// TIA Portal V20 export
DATA_BLOCK "HmiInterface"   // DB95
{ DB_Accessible_From_OPC_UA := 'FALSE' }
AUTHOR : ERsystem_FA2_DH. Kim
// stored: Access Published, DBAccessibleFromOPCUA false, DBAccessibleFromWebserver false, MemoryReserve 100, Namespace Unit1.Em3
   VAR
      em : "LAF_typeEmInterface";
      cm : Struct
         softCam : "Unit1.type_emRelations_em3_SoftCam";
      END_STRUCT;
      webGuide : Struct
         jobs { S7_SetPoint := 'True'} : "LAF_typeJobsInterface";
         sequence { S7_SetPoint := 'True'} : "LAF_typeSequenceInterface";
      END_STRUCT;
      auxiliary : Struct
         cmEpc_UnUse : Bool;
         dancerRegulator : LReal;
      END_STRUCT;
      cmSafetyPinIdlePositionSensor { S7_SetPoint := 'True'} : "LBC_typeDigitalSignalInterface";
      cmRotationSafetyPinPositionSensor { S7_SetPoint := 'True'} : "LBC_typeDigitalSignalInterface";
      cmIonizerTopMaintDetection { S7_SetPoint := 'True'} : "LBC_typeDigitalSignalInterface";
      cmIonizerTopErrorDetection { S7_SetPoint := 'True'} : "LBC_typeDigitalSignalInterface";
      cmIonizerBtmMaintDetection { S7_SetPoint := 'True'} : "LBC_typeDigitalSignalInterface";
      cmIonizerBtmErrorDetection { S7_SetPoint := 'True'} : "LBC_typeDigitalSignalInterface";
      cmDancerEncoder : "LBC_typeAnalogInputInterface";
      cmLoadCellControllerInterface : "LBC_typeAnalogInputInterface";
      cmDancerElectroPneumaticRegulator : "LBC_typeAnalogOutputInterface";
      cmCompensatorAxisX : "LBC_typeAxis64PosInterface";
      cmMasterVirtualAxis { S7_SetPoint := 'True'} : "LBC_typeAxis64PosInterface";
      cmUnwinderVirtualAxis : "LBC_typeAxis64PosInterface";
      cmDancerFwdBwd : "LBC_typeTwoWayActuatorInterface";
      cmSepaUnwinderIonizerTop { S7_SetPoint := 'True'} : "LBC_typeTwoWayActuatorInterface";
      cmSepaUnwinderIonizerBottom { S7_SetPoint := 'True'} : "LBC_typeTwoWayActuatorInterface";
      cmEpcPivot : "LER_typeCON600Interface";
      motion : Struct
         jobs { S7_SetPoint := 'True'} : "LAF_typeJobsInterface";
         sequence { S7_SetPoint := 'True'} : "LAF_typeSequenceInterface";
      END_STRUCT;
      "step" : Struct
         jobs { S7_SetPoint := 'True'} : "LAF_typeJobsInterface";
         sequence { S7_SetPoint := 'True'} : "LAF_typeSequenceInterface";
      END_STRUCT;
      intCondition : Struct
         Axis_03 { S7_SetPoint := 'True'} : "LER.typeAxisIntlockAll";   // compenastor X
         Actuator_10 { S7_SetPoint := 'True'} : "LER.typeAxisActuatorCondition";   // DancerFwdBwd
         Actuator_11 { S7_SetPoint := 'True'} : "LER.typeAxisActuatorCondition";   // SepaUnwinderIonizer
         Actuator_12 { S7_SetPoint := 'True'} : "LER.typeAxisActuatorCondition";   // SepaUnwinderIonizerBottom
      END_STRUCT;
   END_VAR
BEGIN
   em.interlinkMode.link := FALSE;
   em.interlinkMode.unlink := FALSE;
   em.interlinkMode.isLinked := TRUE;
   em.commands.enable := FALSE;
   em.commands.acknowledge := FALSE;
   em.commands.disableAlarms := FALSE;
   em.commands.activateSimulation := FALSE;
   em.commands.home := FALSE;
   em.commands.moveToInitialPosition := FALSE;
   em.commands.directModeControl := 16#0000_0002;
   em.commands.directStateControl := 16#0000_0002;
   em.status.enabled := TRUE;
   em.status.acknowledgeActive := FALSE;
   em.status.alarmsDisabled := FALSE;
   em.status.simulationActive := FALSE;
   em.status.safetyReleased := TRUE;
   em.status.initialized := FALSE;
   em.status.homed := TRUE;
   em.status.safeState := FALSE;
   em.status.stateComplete := TRUE;
   cmSafetyPinIdlePositionSensor.commands.refreshConfiguration := FALSE;
   cmSafetyPinIdlePositionSensor.commands.editConfiguration := FALSE;
   cmSafetyPinIdlePositionSensor.commands.saveConfiguration := FALSE;
   cmSafetyPinIdlePositionSensor.commands.reset := FALSE;
   cmSafetyPinIdlePositionSensor.monitoring.enable := TRUE;
   cmSafetyPinIdlePositionSensor.monitoring.referenceDesignator := WSTRING#'U1.EM3 WebGuide.DigitalSignal';
   cmSafetyPinIdlePositionSensor.monitoring.simulation := FALSE;
   cmSafetyPinIdlePositionSensor.monitoring.processValue := TRUE;
   cmSafetyPinIdlePositionSensor.monitoring.error := FALSE;
   cmSafetyPinIdlePositionSensor.monitoring.status := 16#0000;
   cmSafetyPinIdlePositionSensor.configuration.referenceDesignator := WSTRING#'DigitalSignal';
   cmSafetyPinIdlePositionSensor.configuration.onDelay := T#0MS;
   cmSafetyPinIdlePositionSensor.configuration.offDelay := T#0MS;
   cmSafetyPinIdlePositionSensor.configuration.default := FALSE;
   cmSafetyPinIdlePositionSensor.configuration.invertProcessValue := FALSE;
   cmSafetyPinIdlePositionSensor.configuration.disableAlarms := FALSE;
   cmRotationSafetyPinPositionSensor.commands.refreshConfiguration := FALSE;
   cmRotationSafetyPinPositionSensor.commands.editConfiguration := FALSE;
   cmRotationSafetyPinPositionSensor.commands.saveConfiguration := FALSE;
   cmRotationSafetyPinPositionSensor.commands.reset := FALSE;
   cmRotationSafetyPinPositionSensor.monitoring.enable := TRUE;
   cmRotationSafetyPinPositionSensor.monitoring.referenceDesignator := WSTRING#'U1.EM3 WebGuide.DigitalSignal';
   cmRotationSafetyPinPositionSensor.monitoring.simulation := FALSE;
   cmRotationSafetyPinPositionSensor.monitoring.processValue := TRUE;
   cmRotationSafetyPinPositionSensor.monitoring.error := FALSE;
   cmRotationSafetyPinPositionSensor.monitoring.status := 16#0000;
   cmRotationSafetyPinPositionSensor.configuration.referenceDesignator := WSTRING#'DigitalSignal';
   cmRotationSafetyPinPositionSensor.configuration.onDelay := T#0MS;
   cmRotationSafetyPinPositionSensor.configuration.offDelay := T#0MS;
   cmRotationSafetyPinPositionSensor.configuration.default := FALSE;
   cmRotationSafetyPinPositionSensor.configuration.invertProcessValue := FALSE;
   cmRotationSafetyPinPositionSensor.configuration.disableAlarms := FALSE;
   cmIonizerTopMaintDetection.commands.refreshConfiguration := FALSE;
   cmIonizerTopMaintDetection.commands.editConfiguration := FALSE;
   cmIonizerTopMaintDetection.commands.saveConfiguration := FALSE;
   cmIonizerTopMaintDetection.commands.reset := FALSE;
   cmIonizerTopMaintDetection.monitoring.enable := TRUE;
   cmIonizerTopMaintDetection.monitoring.referenceDesignator := WSTRING#'U1.EM3 WebGuide.DigitalSignal';
   cmIonizerTopMaintDetection.monitoring.simulation := FALSE;
   cmIonizerTopMaintDetection.monitoring.processValue := FALSE;
   cmIonizerTopMaintDetection.monitoring.error := FALSE;
   cmIonizerTopMaintDetection.monitoring.status := 16#0000;
   cmIonizerTopMaintDetection.configuration.referenceDesignator := WSTRING#'DigitalSignal';
   cmIonizerTopMaintDetection.configuration.onDelay := T#0MS;
   cmIonizerTopMaintDetection.configuration.offDelay := T#0MS;
   cmIonizerTopMaintDetection.configuration.default := FALSE;
   cmIonizerTopMaintDetection.configuration.invertProcessValue := FALSE;
   cmIonizerTopMaintDetection.configuration.disableAlarms := FALSE;
   cmIonizerTopErrorDetection.commands.refreshConfiguration := FALSE;
   cmIonizerTopErrorDetection.commands.editConfiguration := FALSE;
   cmIonizerTopErrorDetection.commands.saveConfiguration := FALSE;
   cmIonizerTopErrorDetection.commands.reset := FALSE;
   cmIonizerTopErrorDetection.monitoring.enable := TRUE;
   cmIonizerTopErrorDetection.monitoring.referenceDesignator := WSTRING#'U1.EM3 WebGuide.DigitalSignal';
   cmIonizerTopErrorDetection.monitoring.simulation := FALSE;
   cmIonizerTopErrorDetection.monitoring.processValue := TRUE;
   cmIonizerTopErrorDetection.monitoring.error := FALSE;
   cmIonizerTopErrorDetection.monitoring.status := 16#0000;
   cmIonizerTopErrorDetection.configuration.referenceDesignator := WSTRING#'DigitalSignal';
   cmIonizerTopErrorDetection.configuration.onDelay := T#0MS;
   cmIonizerTopErrorDetection.configuration.offDelay := T#0MS;
   cmIonizerTopErrorDetection.configuration.default := FALSE;
   cmIonizerTopErrorDetection.configuration.invertProcessValue := FALSE;
   cmIonizerTopErrorDetection.configuration.disableAlarms := FALSE;
   cmIonizerBtmMaintDetection.commands.refreshConfiguration := FALSE;
   cmIonizerBtmMaintDetection.commands.editConfiguration := FALSE;
   cmIonizerBtmMaintDetection.commands.saveConfiguration := FALSE;
   cmIonizerBtmMaintDetection.commands.reset := FALSE;
   cmIonizerBtmMaintDetection.monitoring.enable := TRUE;
   cmIonizerBtmMaintDetection.monitoring.referenceDesignator := WSTRING#'U1.EM3 WebGuide.DigitalSignal';
   cmIonizerBtmMaintDetection.monitoring.simulation := FALSE;
   cmIonizerBtmMaintDetection.monitoring.processValue := FALSE;
   cmIonizerBtmMaintDetection.monitoring.error := FALSE;
   cmIonizerBtmMaintDetection.monitoring.status := 16#0000;
   cmIonizerBtmMaintDetection.configuration.referenceDesignator := WSTRING#'DigitalSignal';
   cmIonizerBtmMaintDetection.configuration.onDelay := T#0MS;
   cmIonizerBtmMaintDetection.configuration.offDelay := T#0MS;
   cmIonizerBtmMaintDetection.configuration.default := FALSE;
   cmIonizerBtmMaintDetection.configuration.invertProcessValue := FALSE;
   cmIonizerBtmMaintDetection.configuration.disableAlarms := FALSE;
   cmIonizerBtmErrorDetection.commands.refreshConfiguration := FALSE;
   cmIonizerBtmErrorDetection.commands.editConfiguration := FALSE;
   cmIonizerBtmErrorDetection.commands.saveConfiguration := FALSE;
   cmIonizerBtmErrorDetection.commands.reset := FALSE;
   cmIonizerBtmErrorDetection.monitoring.enable := TRUE;
   cmIonizerBtmErrorDetection.monitoring.referenceDesignator := WSTRING#'U1.EM3 WebGuide.DigitalSignal';
   cmIonizerBtmErrorDetection.monitoring.simulation := FALSE;
   cmIonizerBtmErrorDetection.monitoring.processValue := TRUE;
   cmIonizerBtmErrorDetection.monitoring.error := FALSE;
   cmIonizerBtmErrorDetection.monitoring.status := 16#0000;
   cmIonizerBtmErrorDetection.configuration.referenceDesignator := WSTRING#'DigitalSignal';
   cmIonizerBtmErrorDetection.configuration.onDelay := T#0MS;
   cmIonizerBtmErrorDetection.configuration.offDelay := T#0MS;
   cmIonizerBtmErrorDetection.configuration.default := FALSE;
   cmIonizerBtmErrorDetection.configuration.invertProcessValue := FALSE;
   cmIonizerBtmErrorDetection.configuration.disableAlarms := FALSE;
   cmDancerEncoder.commands.refreshConfiguration := FALSE;
   cmDancerEncoder.commands.editConfiguration := FALSE;
   cmDancerEncoder.commands.saveConfiguration := FALSE;
   cmDancerEncoder.commands.reset := FALSE;
   cmDancerEncoder.monitoring.enable := TRUE;
   cmDancerEncoder.monitoring.referenceDesignator := WSTRING#'U1.EM3 WebGuide.cmDancerEncoder';
   cmDancerEncoder.monitoring.simulation := FALSE;
   cmDancerEncoder.monitoring.processValue := 0.034215856481481;
   cmDancerEncoder.monitoring.analogValue := 13835;
   cmDancerEncoder.monitoring.limitHigh2 := FALSE;
   cmDancerEncoder.monitoring.limitHigh1 := FALSE;
   cmDancerEncoder.monitoring.limitLow1 := FALSE;
   cmDancerEncoder.monitoring.limitLow2 := FALSE;
   cmDancerEncoder.monitoring.maxValueReached := FALSE;
   cmDancerEncoder.monitoring.minValueReached := FALSE;
   cmDancerEncoder.monitoring.error := FALSE;
   cmDancerEncoder.monitoring.status := 16#0000;
   cmDancerEncoder.configuration.referenceDesignator := WSTRING#'cmDancerEncoder';
   cmDancerEncoder.configuration.physicalUnit := 'unit';
   cmDancerEncoder.configuration.isUnipolarSignal := TRUE;
   cmDancerEncoder.configuration.default := 0.0;
   cmDancerEncoder.configuration.limitHigh2 := 20.0;
   cmDancerEncoder.configuration.limitHigh1 := 15.0;
   cmDancerEncoder.configuration.limitLow1 := -15.0;
   cmDancerEncoder.configuration.limitLow2 := -20.0;
   cmDancerEncoder.configuration.processValueMax := 43.0;
   cmDancerEncoder.configuration.processValueMin := -43.0;
   cmDancerEncoder.configuration.scaleAnalogUppPoint := 27648.0;
   cmDancerEncoder.configuration.scaleAnalogLowPoint := 0.0;
   cmDancerEncoder.configuration.scaleProcessUppPoint := 43.0;
   cmDancerEncoder.configuration.scaleProcessLowPoint := -43.0;
   cmDancerEncoder.configuration.disableAlarms := FALSE;
   cmLoadCellControllerInterface.commands.refreshConfiguration := FALSE;
   cmLoadCellControllerInterface.commands.editConfiguration := FALSE;
   cmLoadCellControllerInterface.commands.saveConfiguration := FALSE;
   cmLoadCellControllerInterface.commands.reset := FALSE;
   cmLoadCellControllerInterface.monitoring.enable := TRUE;
   cmLoadCellControllerInterface.monitoring.referenceDesignator := WSTRING#'U1.EM3 WebGuide.cmLoadCellController';
   cmLoadCellControllerInterface.monitoring.simulation := FALSE;
   cmLoadCellControllerInterface.monitoring.processValue := -99.9638310185185;
   cmLoadCellControllerInterface.monitoring.analogValue := 5;
   cmLoadCellControllerInterface.monitoring.limitHigh2 := FALSE;
   cmLoadCellControllerInterface.monitoring.limitHigh1 := FALSE;
   cmLoadCellControllerInterface.monitoring.limitLow1 := TRUE;
   cmLoadCellControllerInterface.monitoring.limitLow2 := TRUE;
   cmLoadCellControllerInterface.monitoring.maxValueReached := FALSE;
   cmLoadCellControllerInterface.monitoring.minValueReached := FALSE;
   cmLoadCellControllerInterface.monitoring.error := FALSE;
   cmLoadCellControllerInterface.monitoring.status := 16#0000;
   cmLoadCellControllerInterface.configuration.referenceDesignator := WSTRING#'cmLoadCellController';
   cmLoadCellControllerInterface.configuration.physicalUnit := 'unit';
   cmLoadCellControllerInterface.configuration.isUnipolarSignal := TRUE;
   cmLoadCellControllerInterface.configuration.default := 0.0;
   cmLoadCellControllerInterface.configuration.limitHigh2 := 90.0;
   cmLoadCellControllerInterface.configuration.limitHigh1 := 80.0;
   cmLoadCellControllerInterface.configuration.limitLow1 := -80.0;
   cmLoadCellControllerInterface.configuration.limitLow2 := -90.0;
   cmLoadCellControllerInterface.configuration.processValueMax := 100.0;
   cmLoadCellControllerInterface.configuration.processValueMin := -100.0;
   cmLoadCellControllerInterface.configuration.scaleAnalogUppPoint := 27648.0;
   cmLoadCellControllerInterface.configuration.scaleAnalogLowPoint := 0.0;
   cmLoadCellControllerInterface.configuration.scaleProcessUppPoint := 100.0;
   cmLoadCellControllerInterface.configuration.scaleProcessLowPoint := -100.0;
   cmLoadCellControllerInterface.configuration.disableAlarms := TRUE;
   cmDancerElectroPneumaticRegulator.commands.refreshConfiguration := FALSE;
   cmDancerElectroPneumaticRegulator.commands.editConfiguration := FALSE;
   cmDancerElectroPneumaticRegulator.commands.saveConfiguration := FALSE;
   cmDancerElectroPneumaticRegulator.commands.reset := FALSE;
   cmDancerElectroPneumaticRegulator.monitoring.enable := TRUE;
   cmDancerElectroPneumaticRegulator.monitoring.referenceDesignator := WSTRING#'cmDancerRegulator';
   cmDancerElectroPneumaticRegulator.monitoring.simulation := FALSE;
   cmDancerElectroPneumaticRegulator.monitoring.processValue := 0.0;
   cmDancerElectroPneumaticRegulator.monitoring.analogValue := 0;
   cmDancerElectroPneumaticRegulator.monitoring.limitHigh2 := FALSE;
   cmDancerElectroPneumaticRegulator.monitoring.limitHigh1 := FALSE;
   cmDancerElectroPneumaticRegulator.monitoring.limitLow1 := TRUE;
   cmDancerElectroPneumaticRegulator.monitoring.limitLow2 := TRUE;
   cmDancerElectroPneumaticRegulator.monitoring.maxValueReached := FALSE;
   cmDancerElectroPneumaticRegulator.monitoring.minValueReached := FALSE;
   cmDancerElectroPneumaticRegulator.monitoring.error := FALSE;
   cmDancerElectroPneumaticRegulator.monitoring.status := 16#0000;
   cmDancerElectroPneumaticRegulator.configuration.referenceDesignator := WSTRING#'cmDancerRegulator';
   cmDancerElectroPneumaticRegulator.configuration.physicalUnit := 'unit';
   cmDancerElectroPneumaticRegulator.configuration.isUnipolarSignal := TRUE;
   cmDancerElectroPneumaticRegulator.configuration.default := 0;
   cmDancerElectroPneumaticRegulator.configuration.limitHigh2 := 0.5;
   cmDancerElectroPneumaticRegulator.configuration.limitHigh1 := 0.5;
   cmDancerElectroPneumaticRegulator.configuration.limitLow1 := 0.0;
   cmDancerElectroPneumaticRegulator.configuration.limitLow2 := 0.0;
   cmDancerElectroPneumaticRegulator.configuration.processValueMax := 0.5;
   cmDancerElectroPneumaticRegulator.configuration.processValueMin := 0.0;
   cmDancerElectroPneumaticRegulator.configuration.scaleProcessUppPoint := 0.5;
   cmDancerElectroPneumaticRegulator.configuration.scaleProcessLowPoint := 0.0;
   cmDancerElectroPneumaticRegulator.configuration.scaleAnalogUppPoint := 27648.0;
   cmDancerElectroPneumaticRegulator.configuration.scaleAnalogLowPoint := 0.0;
   cmDancerElectroPneumaticRegulator.configuration.disableAlarms := TRUE;
   cmCompensatorAxisX.commandConfiguration.generalSettings.stopOnError := TRUE;
   cmCompensatorAxisX.commandConfiguration.generalSettings.resetWithRestart := FALSE;
   cmCompensatorAxisX.commandConfiguration.generalSettings.abortWaitingSyncCmd := TRUE;
   cmCompensatorAxisX.commandConfiguration.power.startMode := 1;
   cmCompensatorAxisX.commandConfiguration.power.stopMode := 0;
   cmCompensatorAxisX.commandConfiguration.power.syncMotionSimulation := FALSE;
   cmCompensatorAxisX.commandConfiguration.power.syncMotionSimulationExtendedMode := -1;
   cmCompensatorAxisX.commandConfiguration.jog.velocity := 10.0;
   cmCompensatorAxisX.commandConfiguration.jog.acceleration := 100.0;
   cmCompensatorAxisX.commandConfiguration.jog.deceleration := 100.0;
   cmCompensatorAxisX.commandConfiguration.jog.jerk := -1.0;
   cmCompensatorAxisX.commandConfiguration.jog.positionControlled := TRUE;
   cmCompensatorAxisX.commandConfiguration.jog.increment := 0.0;
   cmCompensatorAxisX.commandConfiguration.jog.mode := 0;
   cmCompensatorAxisX.commandConfiguration.moveVelocity.velocity := 10.0;
   cmCompensatorAxisX.commandConfiguration.moveVelocity.acceleration := 100.0;
   cmCompensatorAxisX.commandConfiguration.moveVelocity.deceleration := 100.0;
   cmCompensatorAxisX.commandConfiguration.moveVelocity.jerk := -1.0;
   cmCompensatorAxisX.commandConfiguration.moveVelocity.direction := 0;
   cmCompensatorAxisX.commandConfiguration.moveVelocity.positionControlled := TRUE;
   cmCompensatorAxisX.commandConfiguration.moveVelocity.velocityChangeOnTheFly := FALSE;
   cmCompensatorAxisX.commandConfiguration.stop.deceleration := -1.0;
   cmCompensatorAxisX.commandConfiguration.stop.jerk := -1.0;
   cmCompensatorAxisX.commandConfiguration.stop.abortAcceleration := FALSE;
   cmCompensatorAxisX.commandConfiguration.fastStop.deceleration := -1.0;
   cmCompensatorAxisX.commandConfiguration.fastStop.jerk := -1.0;
   cmCompensatorAxisX.commandConfiguration.fastStop.abortAcceleration := FALSE;
   cmCompensatorAxisX.commandConfiguration.fastStop.replaceStopPossible := FALSE;
   cmCompensatorAxisX.commandConfiguration.torqueLimiting.limit := -1.0;
   cmCompensatorAxisX.commandConfiguration.torqueLimiting.mode := 0;
   cmCompensatorAxisX.commandConfiguration.homing.position := 0.0;
   cmCompensatorAxisX.commandConfiguration.homing.mode := 0;
   cmCompensatorAxisX.commandConfiguration.homing.sensor := 0;
   cmCompensatorAxisX.commandConfiguration.homing.extendedMode := -1;
   cmCompensatorAxisX.commandConfiguration.homing.extendedModeTorqueLimit := 0.0;
   cmCompensatorAxisX.commandConfiguration.homing.extendedModeTargetPosition := 0.0;
   cmCompensatorAxisX.commandConfiguration.posRelative.distance := 0.0;
   cmCompensatorAxisX.commandConfiguration.posRelative.velocity := 10.0;
   cmCompensatorAxisX.commandConfiguration.posRelative.acceleration := 100.0;
   cmCompensatorAxisX.commandConfiguration.posRelative.deceleration := 100.0;
   cmCompensatorAxisX.commandConfiguration.posRelative.jerk := -1.0;
   cmCompensatorAxisX.commandConfiguration.posRelative.direction := 0;
   cmCompensatorAxisX.commandConfiguration.posAbsolute.position := 0.0;
   cmCompensatorAxisX.commandConfiguration.posAbsolute.velocity := 0.0;
   cmCompensatorAxisX.commandConfiguration.posAbsolute.acceleration := -1.0;
   cmCompensatorAxisX.commandConfiguration.posAbsolute.deceleration := -1.0;
   cmCompensatorAxisX.commandConfiguration.posAbsolute.jerk := 57.5863648889861;
   cmCompensatorAxisX.commandConfiguration.posAbsolute.direction := 1;
   cmCompensatorAxisX.commandConfiguration.posAbsolute.positionChangeOnTheFly := FALSE;
   cmCompensatorAxisX.commandConfiguration.posAbsolute.velocityChangeOnTheFly := FALSE;
   cmCompensatorAxisX.commandConfiguration.posSuperimposed.distance := 150.5;
   cmCompensatorAxisX.commandConfiguration.posSuperimposed.velocityDiff := 53.921568627451;
   cmCompensatorAxisX.commandConfiguration.posSuperimposed.acceleration := 31.7185697808535;
   cmCompensatorAxisX.commandConfiguration.posSuperimposed.deceleration := 31.7185697808535;
   cmCompensatorAxisX.commandConfiguration.posSuperimposed.jerk := 18.6579822240315;
   cmCompensatorAxisX.commandConfiguration.posSuperimposed.direction := 0;
   cmCompensatorAxisX.commandConfiguration.haltSuperimposed.deceleration := -1.0;
   cmCompensatorAxisX.commandConfiguration.haltSuperimposed.jerk := -1.0;
   cmCompensatorAxisX.commandConfiguration.haltSuperimposed.abortAcceleration := FALSE;
   cmCompensatorAxisX.commandConfiguration.gearInRelative.ratioNumerator := 10000;
   cmCompensatorAxisX.commandConfiguration.gearInRelative.ratioDenominator := 10000;
   cmCompensatorAxisX.commandConfiguration.gearInRelative.acceleration := -1.0;
   cmCompensatorAxisX.commandConfiguration.gearInRelative.deceleration := -1.0;
   cmCompensatorAxisX.commandConfiguration.gearInRelative.jerk := -1.0;
   cmCompensatorAxisX.commandConfiguration.gearInRelative.ratioChangeOnTheFly := FALSE;
   cmCompensatorAxisX.commandConfiguration.gearInAbsolute.ratioNumerator := 1;
   cmCompensatorAxisX.commandConfiguration.gearInAbsolute.ratioDenominator := 1;
   cmCompensatorAxisX.commandConfiguration.gearInAbsolute.masterSyncPosition := 0.0;
   cmCompensatorAxisX.commandConfiguration.gearInAbsolute.slaveSyncPosition := 0.0;
   cmCompensatorAxisX.commandConfiguration.gearInAbsolute.syncProfileReference := 1;
   cmCompensatorAxisX.commandConfiguration.gearInAbsolute.masterStartDistance := 0.0;
   cmCompensatorAxisX.commandConfiguration.gearInAbsolute.velocity := -1.0;
   cmCompensatorAxisX.commandConfiguration.gearInAbsolute.acceleration := -1.0;
   cmCompensatorAxisX.commandConfiguration.gearInAbsolute.deceleration := -1.0;
   cmCompensatorAxisX.commandConfiguration.gearInAbsolute.jerk := -1.0;
   cmCompensatorAxisX.commandConfiguration.gearInAbsolute.syncDirection := 1;
   cmCompensatorAxisX.commandConfiguration.gearInAbsolute.ratioChangeOnTheFly := FALSE;
   cmCompensatorAxisX.commandConfiguration.gearInVelocity.continuousUpdate := FALSE;
   cmCompensatorAxisX.commandConfiguration.gearInVelocity.ratioNumerator := 1;
   cmCompensatorAxisX.commandConfiguration.gearInVelocity.ratioDenominator := 1;
   cmCompensatorAxisX.commandConfiguration.gearInVelocity.acceleration := -1.0;
   cmCompensatorAxisX.commandConfiguration.gearInVelocity.deceleration := -1.0;
   cmCompensatorAxisX.commandConfiguration.gearInVelocity.jerk := -1.0;
   cmCompensatorAxisX.commandConfiguration.gearInVelocity.positionControlled := FALSE;
   cmCompensatorAxisX.commandConfiguration.camIn.masterOffset := 0.0;
   cmCompensatorAxisX.commandConfiguration.camIn.slaveOffset := 0.0;
   cmCompensatorAxisX.commandConfiguration.camIn.masterScaling := 1.0;
   cmCompensatorAxisX.commandConfiguration.camIn.slaveScaling := 1.0;
   cmCompensatorAxisX.commandConfiguration.camIn.masterSyncPosition := 0.0;
   cmCompensatorAxisX.commandConfiguration.camIn.syncProfileReference := 2;
   cmCompensatorAxisX.commandConfiguration.camIn.masterStartDistance := 0.0;
   cmCompensatorAxisX.commandConfiguration.camIn.velocity := 179.738562091503;
   cmCompensatorAxisX.commandConfiguration.camIn.acceleration := 176.214276560297;
   cmCompensatorAxisX.commandConfiguration.camIn.deceleration := 176.214276560297;
   cmCompensatorAxisX.commandConfiguration.camIn.jerk := 172.759094666958;
   cmCompensatorAxisX.commandConfiguration.camIn.applicationMode := 0;
   cmCompensatorAxisX.commandConfiguration.camIn.syncDirection := 3;
   cmCompensatorAxisX.commandConfiguration.gearOutCamOut.slavePosition := 0.0;
   cmCompensatorAxisX.commandConfiguration.gearOutCamOut.syncProfileReference := 1;
   cmCompensatorAxisX.commandConfiguration.gearOutCamOut.masterStopDistance := 0.0;
   cmCompensatorAxisX.commandConfiguration.gearOutCamOut.deceleration := -1.0;
   cmCompensatorAxisX.commandConfiguration.gearOutCamOut.jerk := -1.0;
   cmCompensatorAxisX.commandConfiguration.gearOutCamOut.syncOutDirection := 3;
   cmCompensatorAxisX.commandConfiguration.gearOutCamOut.gearOutCamOutMode := -1;
   cmCompensatorAxisX.commandConfiguration.phasing.phaseShift := 301.0;
   cmCompensatorAxisX.commandConfiguration.phasing.velocity := 89.8692810457516;
   cmCompensatorAxisX.commandConfiguration.phasing.acceleration := 88.1071382801487;
   cmCompensatorAxisX.commandConfiguration.phasing.deceleration := 88.1071382801487;
   cmCompensatorAxisX.commandConfiguration.phasing.jerk := 0.0;
   cmCompensatorAxisX.commandConfiguration.phasing.profileReference := 0;
   cmCompensatorAxisX.commandConfiguration.phasing.phasingDistance := 0.0;
   cmCompensatorAxisX.commandConfiguration.phasing.startPosition := 45.0;
   cmCompensatorAxisX.commandConfiguration.phasing.direction := 3;
   cmCompensatorAxisX.commandConfiguration.phasing.phaseAbsolute := FALSE;
   cmCompensatorAxisX.commandConfiguration.phasing.phaseShiftChangeOnTheFly := FALSE;
   cmCompensatorAxisX.commandConfiguration.offset.offset := 0.0;
   cmCompensatorAxisX.commandConfiguration.offset.profileReference := 1;
   cmCompensatorAxisX.commandConfiguration.offset.offsetDistance := 0.0;
   cmCompensatorAxisX.commandConfiguration.offset.startPosition := 0.0;
   cmCompensatorAxisX.commandConfiguration.offset.direction := 3;
   cmCompensatorAxisX.commandConfiguration.offset.offsetAbsolute := TRUE;
   cmCompensatorAxisX.commandConfiguration.offset.offsetChangeOnTheFly := FALSE;
   cmCompensatorAxisX.commands.enableMasterControl := FALSE;
   cmCompensatorAxisX.commands.enableAxis := TRUE;
   cmCompensatorAxisX.commands.resetAxis := FALSE;
   cmCompensatorAxisX.commands.openBrake := FALSE;
   cmCompensatorAxisX.commands.jogForward := FALSE;
   cmCompensatorAxisX.commands.jogBackward := FALSE;
   cmCompensatorAxisX.commands.moveVelocity := FALSE;
   cmCompensatorAxisX.commands.stop := FALSE;
   cmCompensatorAxisX.commands.fastStop := FALSE;
   cmCompensatorAxisX.commands.torqueLimiting := FALSE;
   cmCompensatorAxisX.commands.homing := FALSE;
   cmCompensatorAxisX.commands.posRelative := FALSE;
   cmCompensatorAxisX.commands.posAbsolute := FALSE;
   cmCompensatorAxisX.commands.posSuperimposed := FALSE;
   cmCompensatorAxisX.commands.haltSuperimposed := FALSE;
   cmCompensatorAxisX.commands.selectSetPosition := -1;
   cmCompensatorAxisX.commands.uploadParameters := FALSE;
   cmCompensatorAxisX.commands.refreshConfiguration := FALSE;
   cmCompensatorAxisX.commands.editConfiguration := FALSE;
   cmCompensatorAxisX.commands.saveConfiguration := FALSE;
   cmCompensatorAxisX.commands.uploadCurrentTorque := FALSE;
   cmCompensatorAxisX.commands.reset := FALSE;
   cmCompensatorAxisX.monitoring.enable := TRUE;
   cmCompensatorAxisX.monitoring.referenceDesignator := WSTRING#'U1.EM3 WebGuide.cmCompensatorAxisX';
   cmCompensatorAxisX.monitoring.enabled := TRUE;
   cmCompensatorAxisX.monitoring.enableManualCmds := TRUE;
   cmCompensatorAxisX.monitoring.reset := FALSE;
   cmCompensatorAxisX.monitoring.resetAxis := FALSE;
   cmCompensatorAxisX.monitoring.enableAxis := TRUE;
   cmCompensatorAxisX.monitoring.openBrake := FALSE;
   cmCompensatorAxisX.monitoring.jogBackward := FALSE;
   cmCompensatorAxisX.monitoring.jogForward := FALSE;
   cmCompensatorAxisX.monitoring.moveVelocity := FALSE;
   cmCompensatorAxisX.monitoring.stop := FALSE;
   cmCompensatorAxisX.monitoring.fastStop := FALSE;
   cmCompensatorAxisX.monitoring.torqueLimiting := FALSE;
   cmCompensatorAxisX.monitoring.homing := FALSE;
   cmCompensatorAxisX.monitoring.posRelative := FALSE;
   cmCompensatorAxisX.monitoring.posAbsolute := FALSE;
   cmCompensatorAxisX.monitoring.posSuperimposed := FALSE;
   cmCompensatorAxisX.monitoring.haltSuperimposed := FALSE;
   cmCompensatorAxisX.monitoring.brakeOpened := FALSE;
   cmCompensatorAxisX.monitoring.axisEnabled := TRUE;
   cmCompensatorAxisX.monitoring.resetActive := FALSE;
   cmCompensatorAxisX.monitoring.inVelocity := FALSE;
   cmCompensatorAxisX.monitoring.inLimitation := FALSE;
   cmCompensatorAxisX.monitoring.inClamping := FALSE;
   cmCompensatorAxisX.monitoring.startSync := FALSE;
   cmCompensatorAxisX.monitoring.inSync := FALSE;
   cmCompensatorAxisX.monitoring.inSimulation := FALSE;
   cmCompensatorAxisX.monitoring.jogSelected := FALSE;
   cmCompensatorAxisX.monitoring.moveVelocitySelected := FALSE;
   cmCompensatorAxisX.monitoring.stopSelected := FALSE;
   cmCompensatorAxisX.monitoring.fastStopSelected := FALSE;
   cmCompensatorAxisX.monitoring.torqueLimitingSelected := FALSE;
   cmCompensatorAxisX.monitoring.homingSelected := FALSE;
   cmCompensatorAxisX.monitoring.posRelativeSelected := FALSE;
   cmCompensatorAxisX.monitoring.posAbsoluteSelected := FALSE;
   cmCompensatorAxisX.monitoring.posSuperimposedSelected := FALSE;
   cmCompensatorAxisX.monitoring.haltSuperimposedSelected := FALSE;
   cmCompensatorAxisX.monitoring.commandBusy := FALSE;
   cmCompensatorAxisX.monitoring.commandDone := FALSE;
   cmCompensatorAxisX.monitoring.commandAborted := FALSE;
   cmCompensatorAxisX.monitoring.homingCommandBusy := FALSE;
   cmCompensatorAxisX.monitoring.homingCommandDone := FALSE;
   cmCompensatorAxisX.monitoring.homingCommandAborted := FALSE;
   cmCompensatorAxisX.monitoring.superimposedBusy := FALSE;
   cmCompensatorAxisX.monitoring.superimposedDone := FALSE;
   cmCompensatorAxisX.monitoring.superimposedAborted := FALSE;
   cmCompensatorAxisX.monitoring.selectSetPosition := -1;
   cmCompensatorAxisX.monitoring.selectionController := FALSE;
   cmCompensatorAxisX.monitoring.interlockGeneral := TRUE;
   cmCompensatorAxisX.monitoring.interlockJogForward := TRUE;
   cmCompensatorAxisX.monitoring.interlockJogBackward := TRUE;
   cmCompensatorAxisX.monitoring.interlockWarningGeneral := FALSE;
   cmCompensatorAxisX.monitoring.interlockWarningJogForward := FALSE;
   cmCompensatorAxisX.monitoring.interlockWarningJogBackward := FALSE;
   cmCompensatorAxisX.monitoring.valid := TRUE;
   cmCompensatorAxisX.monitoring.busy := TRUE;
   cmCompensatorAxisX.monitoring.error := FALSE;
   cmCompensatorAxisX.monitoring.status := 16#7002;
   cmCompensatorAxisX.monitoring.subfunctionStatus := 16#0000;
   cmCompensatorAxisX.monitoring.actualPosition := 69.95;
   cmCompensatorAxisX.monitoring.actualSpeed := -0.005;
   cmCompensatorAxisX.monitoring.speedUnit := 1062;
   cmCompensatorAxisX.monitoring.positionUnit := 1013;
   cmCompensatorAxisX.monitoring.axisType := 1;
   cmCompensatorAxisX.monitoring.maxVelocity := 2500.0;
   cmCompensatorAxisX.monitoring.actualCurrent := 0.0;
   cmCompensatorAxisX.monitoring.actualTorque := 0.0;
   cmCompensatorAxisX.monitoring.velocityOverrideEnabled := FALSE;
   cmCompensatorAxisX.monitoring.sinaParaError := FALSE;
   cmCompensatorAxisX.monitoring.sinaParaStatus := 16#0000_0000;
   cmCompensatorAxisX.configuration.referenceDesignator := WSTRING#'cmCompensatorAxisX';
   cmCompensatorAxisX.configuration.disableAlarms := FALSE;
   cmCompensatorAxisX.configuration.masterControlPopUp := TRUE;
   cmCompensatorAxisX.configuration.setPositions[0].position := 0.0;
   cmCompensatorAxisX.configuration.setPositions[1].position := 50.0;
   cmCompensatorAxisX.configuration.setPositions[2].position := 70.0;
   cmCompensatorAxisX.configuration.setPositions[3..15].position := 0.0;
   cmCompensatorAxisX.configuration.setPositions[0].velocity := -1.0;
   cmCompensatorAxisX.configuration.setPositions[1..2].velocity := 30.0;
   cmCompensatorAxisX.configuration.setPositions[3..15].velocity := -1.0;
   cmCompensatorAxisX.configuration.setPositions[0].acceleration := -1.0;
   cmCompensatorAxisX.configuration.setPositions[1..2].acceleration := 30.0;
   cmCompensatorAxisX.configuration.setPositions[3..15].acceleration := -1.0;
   cmCompensatorAxisX.configuration.setPositions[0].deceleration := -1.0;
   cmCompensatorAxisX.configuration.setPositions[1..2].deceleration := 30.0;
   cmCompensatorAxisX.configuration.setPositions[3..15].deceleration := -1.0;
   cmCompensatorAxisX.configuration.setPositions[0..15]."name" := '';
   cmUnwinderVirtualAxis.commandConfiguration.generalSettings.stopOnError := TRUE;
   cmUnwinderVirtualAxis.commandConfiguration.generalSettings.resetWithRestart := FALSE;
   cmUnwinderVirtualAxis.commandConfiguration.generalSettings.abortWaitingSyncCmd := TRUE;
   cmUnwinderVirtualAxis.commandConfiguration.power.startMode := 1;
   cmUnwinderVirtualAxis.commandConfiguration.power.stopMode := 0;
   cmUnwinderVirtualAxis.commandConfiguration.power.syncMotionSimulation := FALSE;
   cmUnwinderVirtualAxis.commandConfiguration.power.syncMotionSimulationExtendedMode := -1;
   cmUnwinderVirtualAxis.commandConfiguration.jog.velocity := 0.0;
   cmUnwinderVirtualAxis.commandConfiguration.jog.acceleration := -1.0;
   cmUnwinderVirtualAxis.commandConfiguration.jog.deceleration := -1.0;
   cmUnwinderVirtualAxis.commandConfiguration.jog.jerk := -1.0;
   cmUnwinderVirtualAxis.commandConfiguration.jog.positionControlled := TRUE;
   cmUnwinderVirtualAxis.commandConfiguration.jog.increment := 0.0;
   cmUnwinderVirtualAxis.commandConfiguration.jog.mode := 0;
   cmUnwinderVirtualAxis.commandConfiguration.moveVelocity.velocity := 0.0;
   cmUnwinderVirtualAxis.commandConfiguration.moveVelocity.acceleration := -1.0;
   cmUnwinderVirtualAxis.commandConfiguration.moveVelocity.deceleration := -1.0;
   cmUnwinderVirtualAxis.commandConfiguration.moveVelocity.jerk := -1.0;
   cmUnwinderVirtualAxis.commandConfiguration.moveVelocity.direction := 0;
   cmUnwinderVirtualAxis.commandConfiguration.moveVelocity.positionControlled := TRUE;
   cmUnwinderVirtualAxis.commandConfiguration.moveVelocity.velocityChangeOnTheFly := FALSE;
   cmUnwinderVirtualAxis.commandConfiguration.stop.deceleration := -1.0;
   cmUnwinderVirtualAxis.commandConfiguration.stop.jerk := -1.0;
   cmUnwinderVirtualAxis.commandConfiguration.stop.abortAcceleration := FALSE;
   cmUnwinderVirtualAxis.commandConfiguration.fastStop.deceleration := -1.0;
   cmUnwinderVirtualAxis.commandConfiguration.fastStop.jerk := -1.0;
   cmUnwinderVirtualAxis.commandConfiguration.fastStop.abortAcceleration := FALSE;
   cmUnwinderVirtualAxis.commandConfiguration.fastStop.replaceStopPossible := FALSE;
   cmUnwinderVirtualAxis.commandConfiguration.torqueLimiting.limit := -1.0;
   cmUnwinderVirtualAxis.commandConfiguration.torqueLimiting.mode := 0;
   cmUnwinderVirtualAxis.commandConfiguration.homing.position := 0.0;
   cmUnwinderVirtualAxis.commandConfiguration.homing.mode := 0;
   cmUnwinderVirtualAxis.commandConfiguration.homing.sensor := 0;
   cmUnwinderVirtualAxis.commandConfiguration.homing.extendedMode := -1;
   cmUnwinderVirtualAxis.commandConfiguration.homing.extendedModeTorqueLimit := 0.0;
   cmUnwinderVirtualAxis.commandConfiguration.homing.extendedModeTargetPosition := 0.0;
   cmUnwinderVirtualAxis.commandConfiguration.posRelative.distance := 0.0;
   cmUnwinderVirtualAxis.commandConfiguration.posRelative.velocity := 0.0;
   cmUnwinderVirtualAxis.commandConfiguration.posRelative.acceleration := -1.0;
   cmUnwinderVirtualAxis.commandConfiguration.posRelative.deceleration := -1.0;
   cmUnwinderVirtualAxis.commandConfiguration.posRelative.jerk := -1.0;
   cmUnwinderVirtualAxis.commandConfiguration.posRelative.direction := 0;
   cmUnwinderVirtualAxis.commandConfiguration.posAbsolute.position := 0.0;
   cmUnwinderVirtualAxis.commandConfiguration.posAbsolute.velocity := 0.0;
   cmUnwinderVirtualAxis.commandConfiguration.posAbsolute.acceleration := -1.0;
   cmUnwinderVirtualAxis.commandConfiguration.posAbsolute.deceleration := -1.0;
   cmUnwinderVirtualAxis.commandConfiguration.posAbsolute.jerk := -1.0;
   cmUnwinderVirtualAxis.commandConfiguration.posAbsolute.direction := 1;
   cmUnwinderVirtualAxis.commandConfiguration.posAbsolute.positionChangeOnTheFly := FALSE;
   cmUnwinderVirtualAxis.commandConfiguration.posAbsolute.velocityChangeOnTheFly := FALSE;
   cmUnwinderVirtualAxis.commandConfiguration.posSuperimposed.distance := 0.0;
   cmUnwinderVirtualAxis.commandConfiguration.posSuperimposed.velocityDiff := -1.0;
   cmUnwinderVirtualAxis.commandConfiguration.posSuperimposed.acceleration := -1.0;
   cmUnwinderVirtualAxis.commandConfiguration.posSuperimposed.deceleration := -1.0;
   cmUnwinderVirtualAxis.commandConfiguration.posSuperimposed.jerk := -1.0;
   cmUnwinderVirtualAxis.commandConfiguration.posSuperimposed.direction := 0;
   cmUnwinderVirtualAxis.commandConfiguration.haltSuperimposed.deceleration := -1.0;
   cmUnwinderVirtualAxis.commandConfiguration.haltSuperimposed.jerk := -1.0;
   cmUnwinderVirtualAxis.commandConfiguration.haltSuperimposed.abortAcceleration := FALSE;
   cmUnwinderVirtualAxis.commandConfiguration.gearInRelative.ratioNumerator := 1;
   cmUnwinderVirtualAxis.commandConfiguration.gearInRelative.ratioDenominator := 1;
   cmUnwinderVirtualAxis.commandConfiguration.gearInRelative.acceleration := -1.0;
   cmUnwinderVirtualAxis.commandConfiguration.gearInRelative.deceleration := -1.0;
   cmUnwinderVirtualAxis.commandConfiguration.gearInRelative.jerk := -1.0;
   cmUnwinderVirtualAxis.commandConfiguration.gearInRelative.ratioChangeOnTheFly := FALSE;
   cmUnwinderVirtualAxis.commandConfiguration.gearInAbsolute.ratioNumerator := 1;
   cmUnwinderVirtualAxis.commandConfiguration.gearInAbsolute.ratioDenominator := 1;
   cmUnwinderVirtualAxis.commandConfiguration.gearInAbsolute.masterSyncPosition := 0.0;
   cmUnwinderVirtualAxis.commandConfiguration.gearInAbsolute.slaveSyncPosition := 0.0;
   cmUnwinderVirtualAxis.commandConfiguration.gearInAbsolute.syncProfileReference := 1;
   cmUnwinderVirtualAxis.commandConfiguration.gearInAbsolute.masterStartDistance := 0.0;
   cmUnwinderVirtualAxis.commandConfiguration.gearInAbsolute.velocity := -1.0;
   cmUnwinderVirtualAxis.commandConfiguration.gearInAbsolute.acceleration := -1.0;
   cmUnwinderVirtualAxis.commandConfiguration.gearInAbsolute.deceleration := -1.0;
   cmUnwinderVirtualAxis.commandConfiguration.gearInAbsolute.jerk := -1.0;
   cmUnwinderVirtualAxis.commandConfiguration.gearInAbsolute.syncDirection := 1;
   cmUnwinderVirtualAxis.commandConfiguration.gearInAbsolute.ratioChangeOnTheFly := FALSE;
   cmUnwinderVirtualAxis.commandConfiguration.gearInVelocity.continuousUpdate := FALSE;
   cmUnwinderVirtualAxis.commandConfiguration.gearInVelocity.ratioNumerator := 1;
   cmUnwinderVirtualAxis.commandConfiguration.gearInVelocity.ratioDenominator := 1;
   cmUnwinderVirtualAxis.commandConfiguration.gearInVelocity.acceleration := -1.0;
   cmUnwinderVirtualAxis.commandConfiguration.gearInVelocity.deceleration := -1.0;
   cmUnwinderVirtualAxis.commandConfiguration.gearInVelocity.jerk := -1.0;
   cmUnwinderVirtualAxis.commandConfiguration.gearInVelocity.positionControlled := FALSE;
   cmUnwinderVirtualAxis.commandConfiguration.camIn.masterOffset := 0.0;
   cmUnwinderVirtualAxis.commandConfiguration.camIn.slaveOffset := 0.0;
   cmUnwinderVirtualAxis.commandConfiguration.camIn.masterScaling := 1.0;
   cmUnwinderVirtualAxis.commandConfiguration.camIn.slaveScaling := 1.0;
   cmUnwinderVirtualAxis.commandConfiguration.camIn.masterSyncPosition := 0.0;
   cmUnwinderVirtualAxis.commandConfiguration.camIn.syncProfileReference := 1;
   cmUnwinderVirtualAxis.commandConfiguration.camIn.masterStartDistance := 0.0;
   cmUnwinderVirtualAxis.commandConfiguration.camIn.velocity := -1.0;
   cmUnwinderVirtualAxis.commandConfiguration.camIn.acceleration := -1.0;
   cmUnwinderVirtualAxis.commandConfiguration.camIn.deceleration := -1.0;
   cmUnwinderVirtualAxis.commandConfiguration.camIn.jerk := -1.0;
   cmUnwinderVirtualAxis.commandConfiguration.camIn.applicationMode := 0;
   cmUnwinderVirtualAxis.commandConfiguration.camIn.syncDirection := 1;
   cmUnwinderVirtualAxis.commandConfiguration.gearOutCamOut.slavePosition := 0.0;
   cmUnwinderVirtualAxis.commandConfiguration.gearOutCamOut.syncProfileReference := 1;
   cmUnwinderVirtualAxis.commandConfiguration.gearOutCamOut.masterStopDistance := 0.0;
   cmUnwinderVirtualAxis.commandConfiguration.gearOutCamOut.deceleration := -1.0;
   cmUnwinderVirtualAxis.commandConfiguration.gearOutCamOut.jerk := -1.0;
   cmUnwinderVirtualAxis.commandConfiguration.gearOutCamOut.syncOutDirection := 3;
   cmUnwinderVirtualAxis.commandConfiguration.gearOutCamOut.gearOutCamOutMode := -1;
   cmUnwinderVirtualAxis.commandConfiguration.phasing.phaseShift := 0.0;
   cmUnwinderVirtualAxis.commandConfiguration.phasing.velocity := -1.0;
   cmUnwinderVirtualAxis.commandConfiguration.phasing.acceleration := -1.0;
   cmUnwinderVirtualAxis.commandConfiguration.phasing.deceleration := -1.0;
   cmUnwinderVirtualAxis.commandConfiguration.phasing.jerk := -1.0;
   cmUnwinderVirtualAxis.commandConfiguration.phasing.profileReference := 0;
   cmUnwinderVirtualAxis.commandConfiguration.phasing.phasingDistance := 0.0;
   cmUnwinderVirtualAxis.commandConfiguration.phasing.startPosition := 0.0;
   cmUnwinderVirtualAxis.commandConfiguration.phasing.direction := 3;
   cmUnwinderVirtualAxis.commandConfiguration.phasing.phaseAbsolute := TRUE;
   cmUnwinderVirtualAxis.commandConfiguration.phasing.phaseShiftChangeOnTheFly := FALSE;
   cmUnwinderVirtualAxis.commandConfiguration.offset.offset := 0.0;
   cmUnwinderVirtualAxis.commandConfiguration.offset.profileReference := 1;
   cmUnwinderVirtualAxis.commandConfiguration.offset.offsetDistance := 0.0;
   cmUnwinderVirtualAxis.commandConfiguration.offset.startPosition := 0.0;
   cmUnwinderVirtualAxis.commandConfiguration.offset.direction := 3;
   cmUnwinderVirtualAxis.commandConfiguration.offset.offsetAbsolute := TRUE;
   cmUnwinderVirtualAxis.commandConfiguration.offset.offsetChangeOnTheFly := FALSE;
   cmUnwinderVirtualAxis.commands.enableMasterControl := FALSE;
   cmUnwinderVirtualAxis.commands.enableAxis := TRUE;
   cmUnwinderVirtualAxis.commands.resetAxis := FALSE;
   cmUnwinderVirtualAxis.commands.openBrake := FALSE;
   cmUnwinderVirtualAxis.commands.jogForward := FALSE;
   cmUnwinderVirtualAxis.commands.jogBackward := FALSE;
   cmUnwinderVirtualAxis.commands.moveVelocity := FALSE;
   cmUnwinderVirtualAxis.commands.stop := FALSE;
   cmUnwinderVirtualAxis.commands.fastStop := FALSE;
   cmUnwinderVirtualAxis.commands.torqueLimiting := FALSE;
   cmUnwinderVirtualAxis.commands.homing := FALSE;
   cmUnwinderVirtualAxis.commands.posRelative := FALSE;
   cmUnwinderVirtualAxis.commands.posAbsolute := FALSE;
   cmUnwinderVirtualAxis.commands.posSuperimposed := FALSE;
   cmUnwinderVirtualAxis.commands.haltSuperimposed := FALSE;
   cmUnwinderVirtualAxis.commands.selectSetPosition := -1;
   cmUnwinderVirtualAxis.commands.uploadParameters := FALSE;
   cmUnwinderVirtualAxis.commands.refreshConfiguration := FALSE;
   cmUnwinderVirtualAxis.commands.editConfiguration := FALSE;
   cmUnwinderVirtualAxis.commands.saveConfiguration := FALSE;
   cmUnwinderVirtualAxis.commands.uploadCurrentTorque := FALSE;
   cmUnwinderVirtualAxis.commands.reset := FALSE;
   cmUnwinderVirtualAxis.monitoring.enable := TRUE;
   cmUnwinderVirtualAxis.monitoring.referenceDesignator := WSTRING#'U1.EM3 WebGuide.Axis64Pos';
   cmUnwinderVirtualAxis.monitoring.enabled := TRUE;
   cmUnwinderVirtualAxis.monitoring.enableManualCmds := TRUE;
   cmUnwinderVirtualAxis.monitoring.reset := FALSE;
   cmUnwinderVirtualAxis.monitoring.resetAxis := FALSE;
   cmUnwinderVirtualAxis.monitoring.enableAxis := TRUE;
   cmUnwinderVirtualAxis.monitoring.openBrake := FALSE;
   cmUnwinderVirtualAxis.monitoring.jogBackward := FALSE;
   cmUnwinderVirtualAxis.monitoring.jogForward := FALSE;
   cmUnwinderVirtualAxis.monitoring.moveVelocity := FALSE;
   cmUnwinderVirtualAxis.monitoring.stop := FALSE;
   cmUnwinderVirtualAxis.monitoring.fastStop := FALSE;
   cmUnwinderVirtualAxis.monitoring.torqueLimiting := FALSE;
   cmUnwinderVirtualAxis.monitoring.homing := FALSE;
   cmUnwinderVirtualAxis.monitoring.posRelative := FALSE;
   cmUnwinderVirtualAxis.monitoring.posAbsolute := FALSE;
   cmUnwinderVirtualAxis.monitoring.posSuperimposed := FALSE;
   cmUnwinderVirtualAxis.monitoring.haltSuperimposed := FALSE;
   cmUnwinderVirtualAxis.monitoring.brakeOpened := FALSE;
   cmUnwinderVirtualAxis.monitoring.axisEnabled := TRUE;
   cmUnwinderVirtualAxis.monitoring.resetActive := FALSE;
   cmUnwinderVirtualAxis.monitoring.inVelocity := FALSE;
   cmUnwinderVirtualAxis.monitoring.inLimitation := FALSE;
   cmUnwinderVirtualAxis.monitoring.inClamping := FALSE;
   cmUnwinderVirtualAxis.monitoring.startSync := FALSE;
   cmUnwinderVirtualAxis.monitoring.inSync := FALSE;
   cmUnwinderVirtualAxis.monitoring.inSimulation := FALSE;
   cmUnwinderVirtualAxis.monitoring.jogSelected := FALSE;
   cmUnwinderVirtualAxis.monitoring.moveVelocitySelected := FALSE;
   cmUnwinderVirtualAxis.monitoring.stopSelected := FALSE;
   cmUnwinderVirtualAxis.monitoring.fastStopSelected := FALSE;
   cmUnwinderVirtualAxis.monitoring.torqueLimitingSelected := FALSE;
   cmUnwinderVirtualAxis.monitoring.homingSelected := FALSE;
   cmUnwinderVirtualAxis.monitoring.posRelativeSelected := FALSE;
   cmUnwinderVirtualAxis.monitoring.posAbsoluteSelected := FALSE;
   cmUnwinderVirtualAxis.monitoring.posSuperimposedSelected := FALSE;
   cmUnwinderVirtualAxis.monitoring.haltSuperimposedSelected := FALSE;
   cmUnwinderVirtualAxis.monitoring.commandBusy := FALSE;
   cmUnwinderVirtualAxis.monitoring.commandDone := FALSE;
   cmUnwinderVirtualAxis.monitoring.commandAborted := FALSE;
   cmUnwinderVirtualAxis.monitoring.homingCommandBusy := FALSE;
   cmUnwinderVirtualAxis.monitoring.homingCommandDone := FALSE;
   cmUnwinderVirtualAxis.monitoring.homingCommandAborted := FALSE;
   cmUnwinderVirtualAxis.monitoring.superimposedBusy := FALSE;
   cmUnwinderVirtualAxis.monitoring.superimposedDone := FALSE;
   cmUnwinderVirtualAxis.monitoring.superimposedAborted := FALSE;
   cmUnwinderVirtualAxis.monitoring.selectSetPosition := -1;
   cmUnwinderVirtualAxis.monitoring.selectionController := FALSE;
   cmUnwinderVirtualAxis.monitoring.interlockGeneral := TRUE;
   cmUnwinderVirtualAxis.monitoring.interlockJogForward := TRUE;
   cmUnwinderVirtualAxis.monitoring.interlockJogBackward := TRUE;
   cmUnwinderVirtualAxis.monitoring.interlockWarningGeneral := FALSE;
   cmUnwinderVirtualAxis.monitoring.interlockWarningJogForward := FALSE;
   cmUnwinderVirtualAxis.monitoring.interlockWarningJogBackward := FALSE;
   cmUnwinderVirtualAxis.monitoring.valid := TRUE;
   cmUnwinderVirtualAxis.monitoring.busy := TRUE;
   cmUnwinderVirtualAxis.monitoring.error := FALSE;
   cmUnwinderVirtualAxis.monitoring.status := 16#7002;
   cmUnwinderVirtualAxis.monitoring.subfunctionStatus := 16#0000;
   cmUnwinderVirtualAxis.monitoring.actualPosition := 0.0;
   cmUnwinderVirtualAxis.monitoring.actualSpeed := 0.0;
   cmUnwinderVirtualAxis.monitoring.speedUnit := 1062;
   cmUnwinderVirtualAxis.monitoring.positionUnit := 1013;
   cmUnwinderVirtualAxis.monitoring.axisType := 1;
   cmUnwinderVirtualAxis.monitoring.maxVelocity := 500.0;
   cmUnwinderVirtualAxis.monitoring.actualCurrent := 0.0;
   cmUnwinderVirtualAxis.monitoring.actualTorque := 0.0;
   cmUnwinderVirtualAxis.monitoring.velocityOverrideEnabled := FALSE;
   cmUnwinderVirtualAxis.monitoring.sinaParaError := FALSE;
   cmUnwinderVirtualAxis.monitoring.sinaParaStatus := 16#0000_0000;
   cmUnwinderVirtualAxis.configuration.referenceDesignator := WSTRING#'Axis64Pos';
   cmUnwinderVirtualAxis.configuration.disableAlarms := TRUE;
   cmUnwinderVirtualAxis.configuration.masterControlPopUp := TRUE;
   cmUnwinderVirtualAxis.configuration.setPositions[0..15].position := 0.0;
   cmUnwinderVirtualAxis.configuration.setPositions[0..15].velocity := -1.0;
   cmUnwinderVirtualAxis.configuration.setPositions[0..15].acceleration := -1.0;
   cmUnwinderVirtualAxis.configuration.setPositions[0..15].deceleration := -1.0;
   cmUnwinderVirtualAxis.configuration.setPositions[0..15]."name" := '';
   cmDancerFwdBwd.commands.refreshConfiguration := FALSE;
   cmDancerFwdBwd.commands.editConfiguration := FALSE;
   cmDancerFwdBwd.commands.saveConfiguration := FALSE;
   cmDancerFwdBwd.commands.reset := FALSE;
   cmDancerFwdBwd.commands.commandHomePos := FALSE;
   cmDancerFwdBwd.commands.commandWorkPos := FALSE;
   cmDancerFwdBwd.monitoring.enable := TRUE;
   cmDancerFwdBwd.monitoring.referenceDesignator := WSTRING#'U1.EM3 WebGuide.cmDancerFwdBwd';
   cmDancerFwdBwd.monitoring.commandHomePos := FALSE;
   cmDancerFwdBwd.monitoring.commandWorkPos := FALSE;
   cmDancerFwdBwd.monitoring.goToHomePos := FALSE;
   cmDancerFwdBwd.monitoring.goToWorkPos := FALSE;
   cmDancerFwdBwd.monitoring.inHomePos := FALSE;
   cmDancerFwdBwd.monitoring.inWorkPos := FALSE;
   cmDancerFwdBwd.monitoring.reset := FALSE;
   cmDancerFwdBwd.monitoring.enableManualCmds := TRUE;
   cmDancerFwdBwd.monitoring.error := FALSE;
   cmDancerFwdBwd.monitoring.interlockHomePos := TRUE;
   cmDancerFwdBwd.monitoring.interlockWorkPos := TRUE;
   cmDancerFwdBwd.monitoring.status := 16#7003;
   cmDancerFwdBwd.monitoring.interlockWarningWorkPos := FALSE;
   cmDancerFwdBwd.monitoring.interlockWarningHomePos := FALSE;
   cmDancerFwdBwd.configuration.referenceDesignator := WSTRING#'cmDancerFwdBwd';
   cmDancerFwdBwd.configuration.monitoringLeavingFeedback := T#1S;
   cmDancerFwdBwd.configuration.monitoringReachingFeedback := T#1S;
   cmDancerFwdBwd.configuration.monitoringDiscrepancy := T#0MS;
   cmDancerFwdBwd.configuration.setOutputHomeContinuously := TRUE;
   cmDancerFwdBwd.configuration.setOutputWorkContinuously := TRUE;
   cmDancerFwdBwd.configuration.disableHomeCommand := FALSE;
   cmDancerFwdBwd.configuration.disableFeedbackHomePos := TRUE;
   cmDancerFwdBwd.configuration.disableFeedbackWorkPos := TRUE;
   cmDancerFwdBwd.configuration.disableAlarms := TRUE;
   cmDancerFwdBwd.configuration.resetOutputsOnError := FALSE;
   cmDancerFwdBwd.configuration.allwaysWaitOnReachingTime := FALSE;
   cmSepaUnwinderIonizerTop.commands.refreshConfiguration := FALSE;
   cmSepaUnwinderIonizerTop.commands.editConfiguration := FALSE;
   cmSepaUnwinderIonizerTop.commands.saveConfiguration := FALSE;
   cmSepaUnwinderIonizerTop.commands.reset := FALSE;
   cmSepaUnwinderIonizerTop.commands.commandHomePos := FALSE;
   cmSepaUnwinderIonizerTop.commands.commandWorkPos := FALSE;
   cmSepaUnwinderIonizerTop.monitoring.enable := TRUE;
   cmSepaUnwinderIonizerTop.monitoring.referenceDesignator := WSTRING#'U1.EM3 WebGuide.cmSepaUnwinderIonizerTop';
   cmSepaUnwinderIonizerTop.monitoring.commandHomePos := FALSE;
   cmSepaUnwinderIonizerTop.monitoring.commandWorkPos := FALSE;
   cmSepaUnwinderIonizerTop.monitoring.goToHomePos := FALSE;
   cmSepaUnwinderIonizerTop.monitoring.goToWorkPos := FALSE;
   cmSepaUnwinderIonizerTop.monitoring.inHomePos := FALSE;
   cmSepaUnwinderIonizerTop.monitoring.inWorkPos := FALSE;
   cmSepaUnwinderIonizerTop.monitoring.reset := FALSE;
   cmSepaUnwinderIonizerTop.monitoring.enableManualCmds := TRUE;
   cmSepaUnwinderIonizerTop.monitoring.error := FALSE;
   cmSepaUnwinderIonizerTop.monitoring.interlockHomePos := TRUE;
   cmSepaUnwinderIonizerTop.monitoring.interlockWorkPos := TRUE;
   cmSepaUnwinderIonizerTop.monitoring.status := 16#7003;
   cmSepaUnwinderIonizerTop.monitoring.interlockWarningWorkPos := FALSE;
   cmSepaUnwinderIonizerTop.monitoring.interlockWarningHomePos := FALSE;
   cmSepaUnwinderIonizerTop.configuration.referenceDesignator := WSTRING#'cmSepaUnwinderIonizerTop';
   cmSepaUnwinderIonizerTop.configuration.monitoringLeavingFeedback := T#5S;
   cmSepaUnwinderIonizerTop.configuration.monitoringReachingFeedback := T#5S;
   cmSepaUnwinderIonizerTop.configuration.monitoringDiscrepancy := T#0MS;
   cmSepaUnwinderIonizerTop.configuration.setOutputHomeContinuously := TRUE;
   cmSepaUnwinderIonizerTop.configuration.setOutputWorkContinuously := TRUE;
   cmSepaUnwinderIonizerTop.configuration.disableHomeCommand := FALSE;
   cmSepaUnwinderIonizerTop.configuration.disableFeedbackHomePos := TRUE;
   cmSepaUnwinderIonizerTop.configuration.disableFeedbackWorkPos := TRUE;
   cmSepaUnwinderIonizerTop.configuration.disableAlarms := FALSE;
   cmSepaUnwinderIonizerTop.configuration.resetOutputsOnError := FALSE;
   cmSepaUnwinderIonizerTop.configuration.allwaysWaitOnReachingTime := FALSE;
   cmSepaUnwinderIonizerBottom.commands.refreshConfiguration := FALSE;
   cmSepaUnwinderIonizerBottom.commands.editConfiguration := FALSE;
   cmSepaUnwinderIonizerBottom.commands.saveConfiguration := FALSE;
   cmSepaUnwinderIonizerBottom.commands.reset := FALSE;
   cmSepaUnwinderIonizerBottom.commands.commandHomePos := FALSE;
   cmSepaUnwinderIonizerBottom.commands.commandWorkPos := FALSE;
   cmSepaUnwinderIonizerBottom.monitoring.enable := TRUE;
   cmSepaUnwinderIonizerBottom.monitoring.referenceDesignator := WSTRING#'U1.EM3 WebGuide.cmSepaUnwinderIonizerBtm';
   cmSepaUnwinderIonizerBottom.monitoring.commandHomePos := FALSE;
   cmSepaUnwinderIonizerBottom.monitoring.commandWorkPos := FALSE;
   cmSepaUnwinderIonizerBottom.monitoring.goToHomePos := FALSE;
   cmSepaUnwinderIonizerBottom.monitoring.goToWorkPos := FALSE;
   cmSepaUnwinderIonizerBottom.monitoring.inHomePos := FALSE;
   cmSepaUnwinderIonizerBottom.monitoring.inWorkPos := FALSE;
   cmSepaUnwinderIonizerBottom.monitoring.reset := FALSE;
   cmSepaUnwinderIonizerBottom.monitoring.enableManualCmds := TRUE;
   cmSepaUnwinderIonizerBottom.monitoring.error := FALSE;
   cmSepaUnwinderIonizerBottom.monitoring.interlockHomePos := TRUE;
   cmSepaUnwinderIonizerBottom.monitoring.interlockWorkPos := TRUE;
   cmSepaUnwinderIonizerBottom.monitoring.status := 16#7003;
   cmSepaUnwinderIonizerBottom.monitoring.interlockWarningWorkPos := FALSE;
   cmSepaUnwinderIonizerBottom.monitoring.interlockWarningHomePos := FALSE;
   cmSepaUnwinderIonizerBottom.configuration.referenceDesignator := WSTRING#'cmSepaUnwinderIonizerBtm';
   cmSepaUnwinderIonizerBottom.configuration.monitoringLeavingFeedback := T#5S;
   cmSepaUnwinderIonizerBottom.configuration.monitoringReachingFeedback := T#5S;
   cmSepaUnwinderIonizerBottom.configuration.monitoringDiscrepancy := T#0MS;
   cmSepaUnwinderIonizerBottom.configuration.setOutputHomeContinuously := TRUE;
   cmSepaUnwinderIonizerBottom.configuration.setOutputWorkContinuously := TRUE;
   cmSepaUnwinderIonizerBottom.configuration.disableHomeCommand := FALSE;
   cmSepaUnwinderIonizerBottom.configuration.disableFeedbackHomePos := TRUE;
   cmSepaUnwinderIonizerBottom.configuration.disableFeedbackWorkPos := TRUE;
   cmSepaUnwinderIonizerBottom.configuration.disableAlarms := FALSE;
   cmSepaUnwinderIonizerBottom.configuration.resetOutputsOnError := FALSE;
   cmSepaUnwinderIonizerBottom.configuration.allwaysWaitOnReachingTime := FALSE;
END_DATA_BLOCK
